(* LS Electric XG5000 project: 241004_인터록 *)
(* PLC LSPLC *)
(* module base 0 slot 0: 입력 모듈:XGI-D21A (DC 24V 입력, 8점 (전류소스/싱크입력)) *)
(* module base 0 slot 1: 출력 모듈:XGQ-RY1A (릴레이 출력, 8점 (2A용, 단독 COM.)) *)

PROGRAM NewProgram (* task: 스캔 프로그램 *)
VAR
    역회전 AT %IX0.0.2 : BOOL;
    역회전램프 AT %QX0.1.1 : BOOL;
    정지 AT %IX0.0.0 : BOOL;
    정회전 AT %IX0.0.1 : BOOL;
    정회전램프 AT %QX0.1.0 : BOOL;
END_VAR

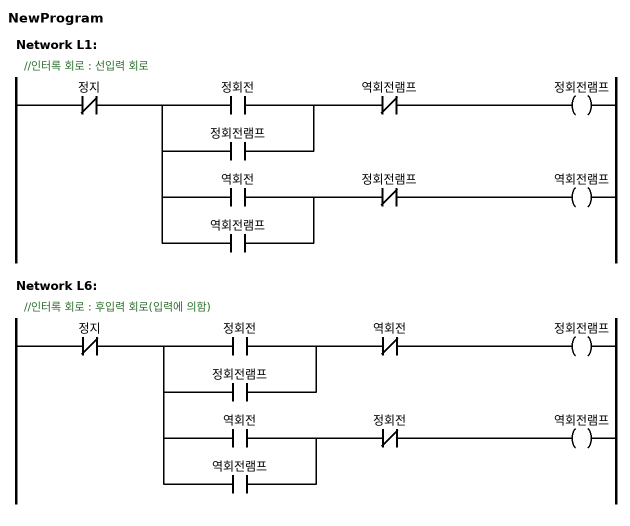
(* //인터록 회로 : 선입력 회로 *)
(* Rung L1 *)
정회전램프 := NOT 정지 AND (정회전 OR 정회전램프) AND NOT 역회전램프;
역회전램프 := NOT 정지 AND (역회전 OR 역회전램프) AND NOT 정회전램프;
(* //인터록 회로 : 후입력 회로(입력에 의함) *)
(* Rung L6 *)
정회전램프 := NOT 정지 AND (정회전 OR 정회전램프) AND NOT 역회전;
역회전램프 := NOT 정지 AND (역회전 OR 역회전램프) AND NOT 정회전;
END_PROGRAM